FUNCTION_BLOCK THROUGH_BLOCK (* Basic FB with empty ECC *)
  (* Standard: 61499-2 *)
  (* Version 1.0, 2026-01-26, obotnar *)
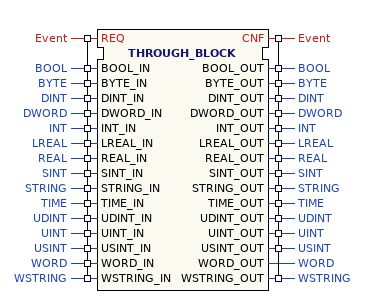
  EVENT_INPUT
    REQ WITH BOOL_IN, BYTE_IN, DINT_IN, DWORD_IN, INT_IN, LREAL_IN, REAL_IN, WSTRING_IN, WORD_IN, USINT_IN, UINT_IN, UDINT_IN, TIME_IN, STRING_IN, SINT_IN;
  END_EVENT
  EVENT_OUTPUT
    CNF WITH WSTRING_OUT, USINT_OUT, UINT_OUT, UDINT_OUT, TIME_OUT, SINT_OUT, BOOL_OUT, BYTE_OUT, DINT_OUT, DWORD_OUT, INT_OUT, LREAL_OUT, REAL_OUT, STRING_OUT;
  END_EVENT
  VAR_INPUT
    BOOL_IN : BOOL;
    BYTE_IN : BYTE;
    DINT_IN : DINT;
    DWORD_IN : DWORD;
    INT_IN : INT;
    LREAL_IN : LREAL;
    REAL_IN : REAL;
    SINT_IN : SINT;
    STRING_IN : STRING;
    TIME_IN : TIME;
    UDINT_IN : UDINT;
    UINT_IN : UINT;
    USINT_IN : USINT;
    WORD_IN : WORD;
    WSTRING_IN : WSTRING;
  END_VAR
  VAR_OUTPUT
    BOOL_OUT : BOOL;
    BYTE_OUT : BYTE;
    DINT_OUT : DINT;
    DWORD_OUT : DWORD;
    INT_OUT : INT;
    LREAL_OUT : LREAL;
    REAL_OUT : REAL;
    SINT_OUT : SINT;
    STRING_OUT : STRING;
    TIME_OUT : TIME;
    UDINT_OUT : UDINT;
    UINT_OUT : UINT;
    USINT_OUT : USINT;
    WORD_OUT : WORD;
    WSTRING_OUT : WSTRING;
  END_VAR
  EC_STATES
    START; (* Initial State *)
  END_STATES
END_FUNCTION_BLOCK
